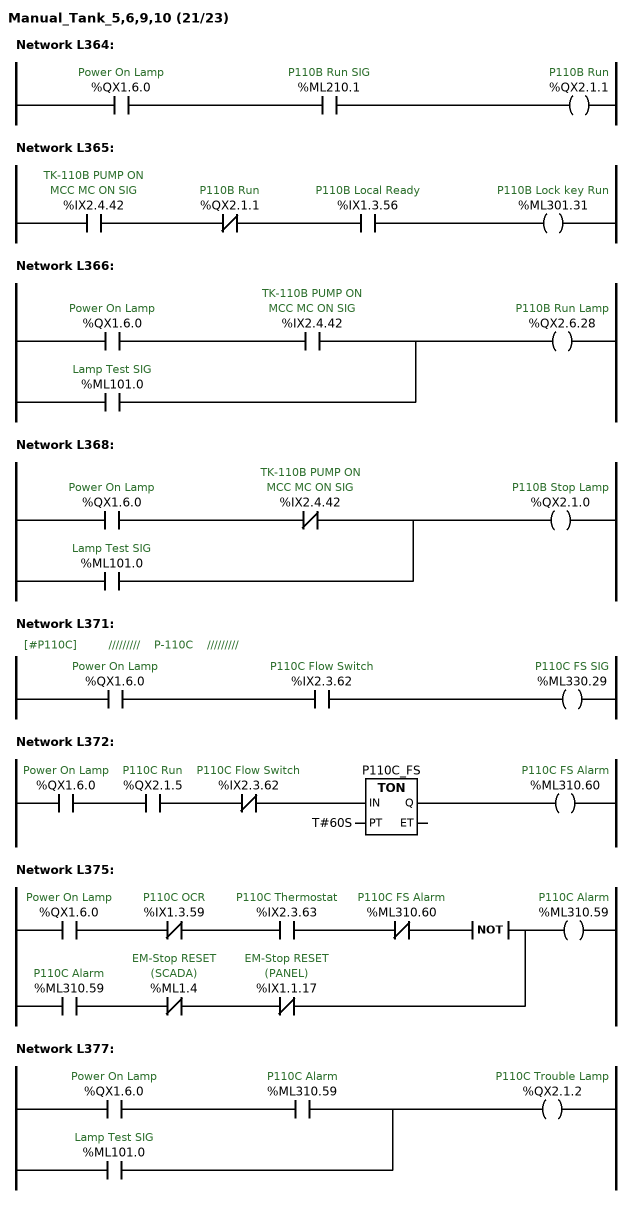
(* [picture p72: Manual_Tank_5,6,9,10 rungs L364-L377] *)
(* Rung L364 *)
%QX2.1.1 := %QX1.6.0 AND %ML210.1;
(* Rung L365 *)
%ML301.31 := %IX2.4.42 AND NOT %QX2.1.1 AND %IX1.3.56;
(* Rung L366 *)
%QX2.6.28 := (%QX1.6.0 AND %IX2.4.42) OR %ML101.0;
(* Rung L368 *)
%QX2.1.0 := (%QX1.6.0 AND NOT %IX2.4.42) OR %ML101.0;
(* [#P110C]         /////////    P-110C    ///////// *)
(* Rung L371 *)
%ML330.29 := %QX1.6.0 AND %IX2.3.62;
(* Rung L372 *)
P110C_FS(IN := %QX1.6.0 AND %QX2.1.5 AND NOT %IX2.3.62, PT := T#60S);
%ML310.60 := P110C_FS.Q;
(* Rung L375 *)
%ML310.59 := NOT (%QX1.6.0 AND NOT %IX1.3.59 AND %IX2.3.63 AND NOT %ML310.60) OR (%ML310.59 AND NOT %ML1.4 AND NOT %IX1.1.17);
(* Rung L377 *)
%QX2.1.2 := (%QX1.6.0 AND %ML310.59) OR %ML101.0;

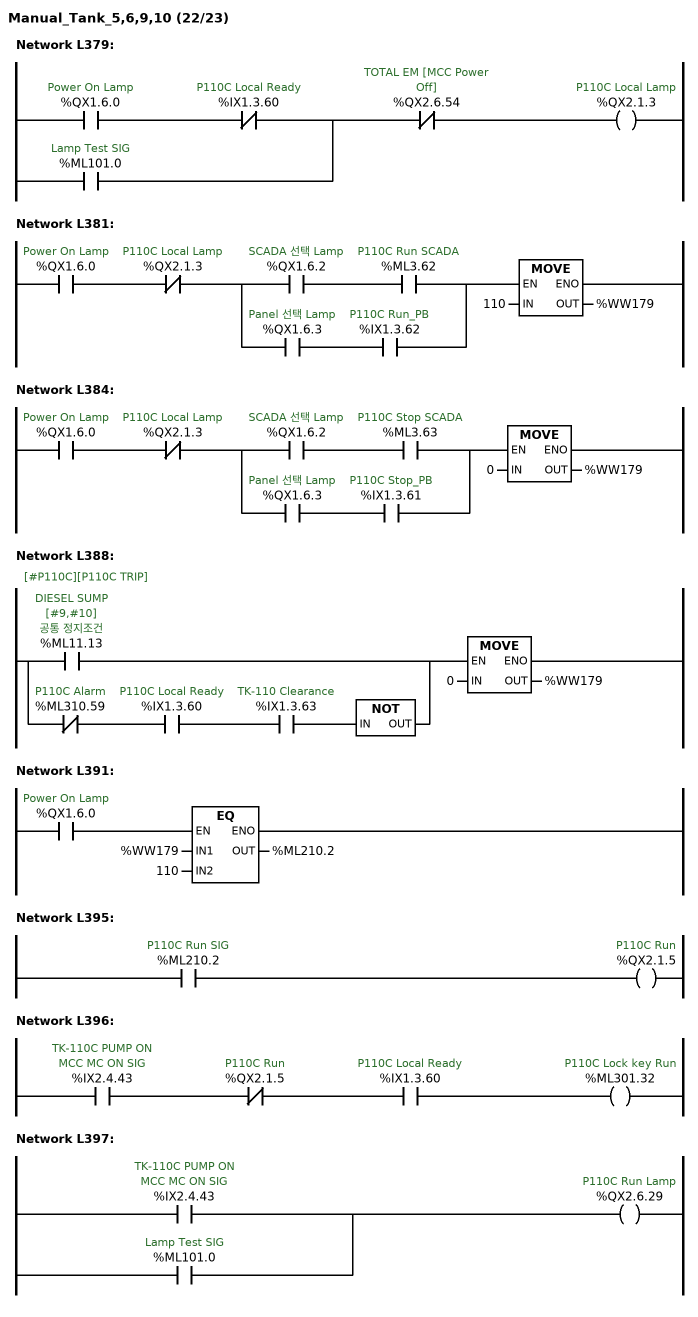
(* Rung L379 *)
%QX2.1.3 := ((%QX1.6.0 AND NOT %IX1.3.60) OR %ML101.0) AND NOT %QX2.6.54;
(* Rung L381 *)
IF %QX1.6.0 AND NOT %QX2.1.3 AND ((%QX1.6.2 AND %ML3.62) OR (%QX1.6.3 AND %IX1.3.62)) THEN
    %WW179 := 110;
END_IF;
(* Rung L384 *)
IF %QX1.6.0 AND NOT %QX2.1.3 AND ((%QX1.6.2 AND %ML3.63) OR (%QX1.6.3 AND %IX1.3.61)) THEN
    %WW179 := 0;
END_IF;
(* [#P110C][P110C TRIP] *)
(* Rung L388 *)
IF %ML11.13 OR (NOT (NOT %ML310.59 AND %IX1.3.60 AND %IX1.3.63)) THEN %WW179 := 0; END_IF;
(* Rung L391 *)
IF %QX1.6.0 THEN %ML210.2 := %WW179 = 110; END_IF;
(* Rung L395 *)
%QX2.1.5 := %ML210.2;
(* Rung L396 *)
%ML301.32 := %IX2.4.43 AND NOT %QX2.1.5 AND %IX1.3.60;
(* Rung L397 *)
%QX2.6.29 := %IX2.4.43 OR %ML101.0;

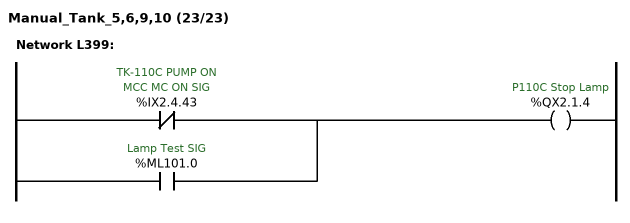
(* Rung L399 *)
%QX2.1.4 := NOT %IX2.4.43 OR %ML101.0;
END_PROGRAM

PROGRAM Manual_Drain_Tank (* task: 스캔 프로그램 *)
VAR
    TK_111_FS : TON;
    TK_112_FS : TON;
    TK_113_FS : TON;
END_VAR

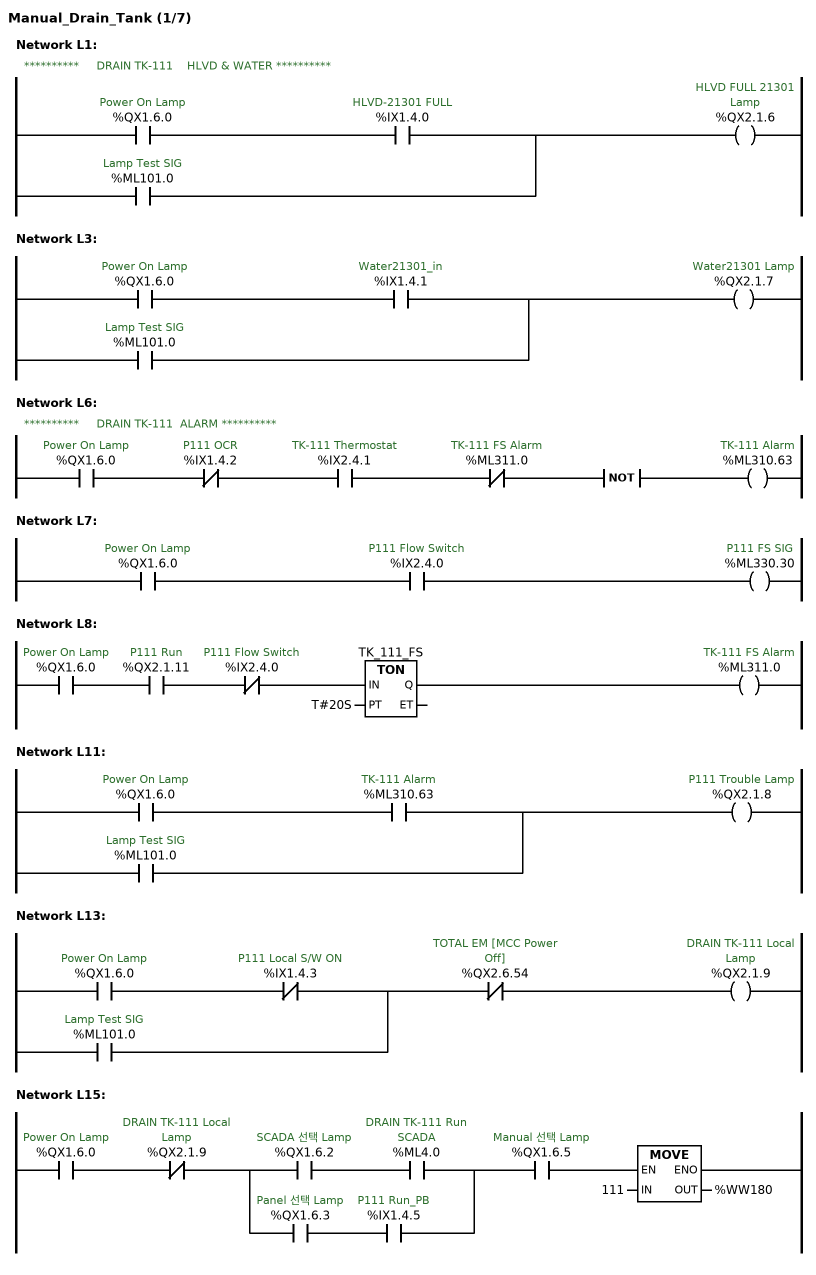
(* **********     DRAIN TK-111    HLVD & WATER ********** *)
(* Rung L1 *)
%QX2.1.6 := (%QX1.6.0 AND %IX1.4.0) OR %ML101.0;
(* Rung L3 *)
%QX2.1.7 := (%QX1.6.0 AND %IX1.4.1) OR %ML101.0;
(* **********     DRAIN TK-111  ALARM ********** *)
(* Rung L6 *)
%ML310.63 := NOT (%QX1.6.0 AND NOT %IX1.4.2 AND %IX2.4.1 AND NOT %ML311.0);
(* Rung L7 *)
%ML330.30 := %QX1.6.0 AND %IX2.4.0;
(* Rung L8 *)
TK_111_FS(IN := %QX1.6.0 AND %QX2.1.11 AND NOT %IX2.4.0, PT := T#20S);
%ML311.0 := TK_111_FS.Q;
(* Rung L11 *)
%QX2.1.8 := (%QX1.6.0 AND %ML310.63) OR %ML101.0;
(* Rung L13 *)
%QX2.1.9 := ((%QX1.6.0 AND NOT %IX1.4.3) OR %ML101.0) AND NOT %QX2.6.54;
(* Rung L15 *)
IF %QX1.6.0 AND NOT %QX2.1.9 AND ((%QX1.6.2 AND %ML4.0) OR (%QX1.6.3 AND %IX1.4.5)) AND %QX1.6.5 THEN
    %WW180 := 111;
END_IF;

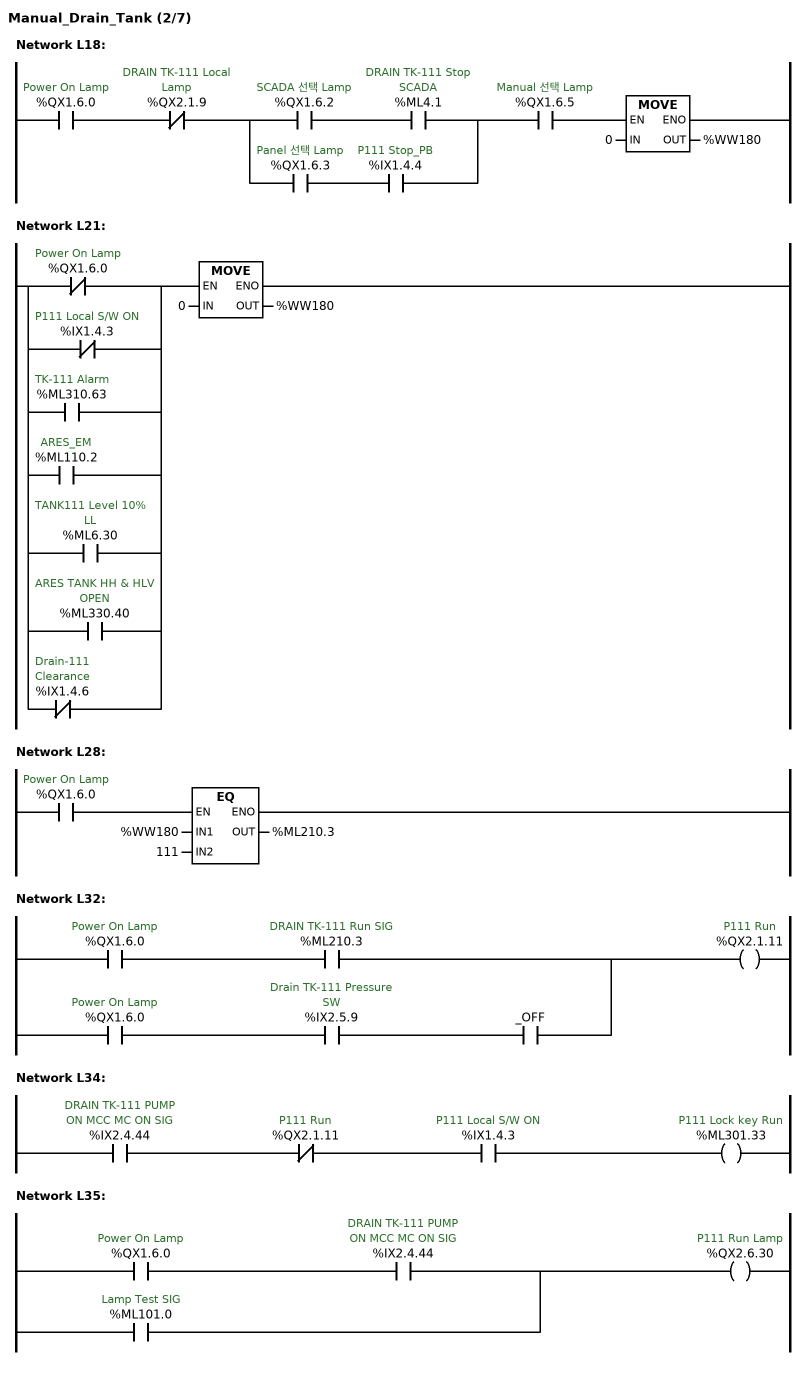
(* Rung L18 *)
IF %QX1.6.0 AND NOT %QX2.1.9 AND ((%QX1.6.2 AND %ML4.1) OR (%QX1.6.3 AND %IX1.4.4)) AND %QX1.6.5 THEN
    %WW180 := 0;
END_IF;
(* Rung L21 *)
IF NOT %QX1.6.0 OR NOT %IX1.4.3 OR %ML310.63 OR %ML110.2 OR %ML6.30 OR %ML330.40 OR NOT %IX1.4.6 THEN
    %WW180 := 0;
END_IF;
(* Rung L28 *)
IF %QX1.6.0 THEN %ML210.3 := %WW180 = 111; END_IF;
(* Rung L32 *)
%QX2.1.11 := (%QX1.6.0 AND %ML210.3) OR (%QX1.6.0 AND %IX2.5.9 AND _OFF);
(* Rung L34 *)
%ML301.33 := %IX2.4.44 AND NOT %QX2.1.11 AND %IX1.4.3;
(* Rung L35 *)
%QX2.6.30 := (%QX1.6.0 AND %IX2.4.44) OR %ML101.0;

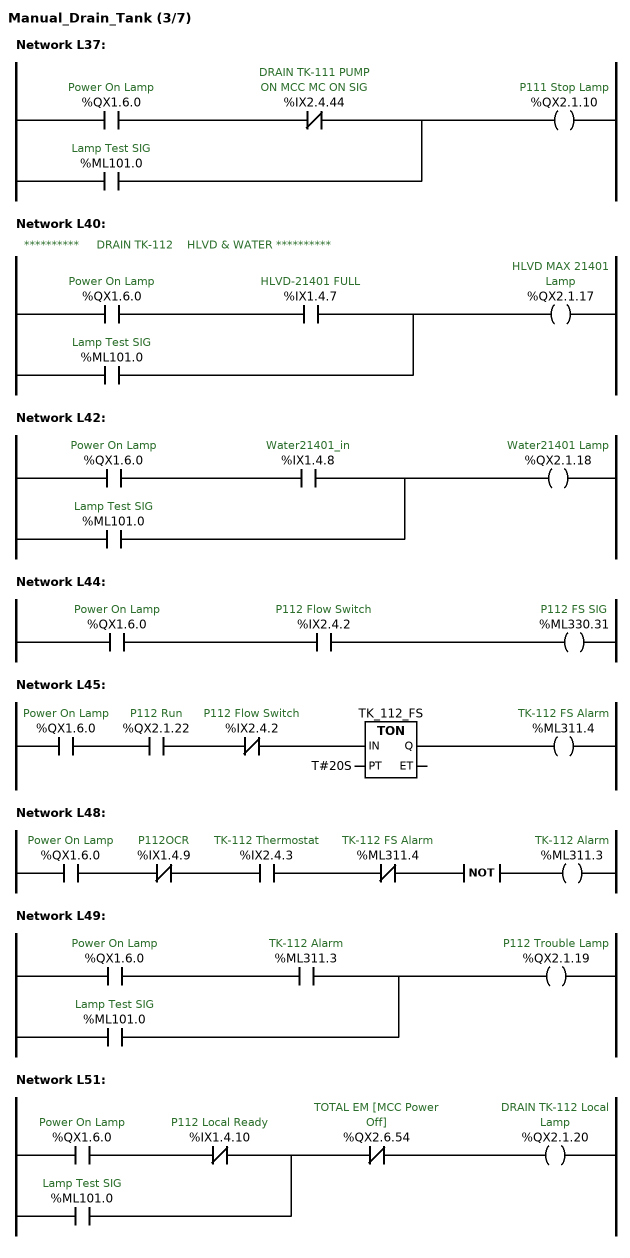
(* Rung L37 *)
%QX2.1.10 := (%QX1.6.0 AND NOT %IX2.4.44) OR %ML101.0;
(* **********     DRAIN TK-112    HLVD & WATER ********** *)
(* Rung L40 *)
%QX2.1.17 := (%QX1.6.0 AND %IX1.4.7) OR %ML101.0;
(* Rung L42 *)
%QX2.1.18 := (%QX1.6.0 AND %IX1.4.8) OR %ML101.0;
(* Rung L44 *)
%ML330.31 := %QX1.6.0 AND %IX2.4.2;
(* Rung L45 *)
TK_112_FS(IN := %QX1.6.0 AND %QX2.1.22 AND NOT %IX2.4.2, PT := T#20S);
%ML311.4 := TK_112_FS.Q;
(* Rung L48 *)
%ML311.3 := NOT (%QX1.6.0 AND NOT %IX1.4.9 AND %IX2.4.3 AND NOT %ML311.4);
(* Rung L49 *)
%QX2.1.19 := (%QX1.6.0 AND %ML311.3) OR %ML101.0;
(* Rung L51 *)
%QX2.1.20 := ((%QX1.6.0 AND NOT %IX1.4.10) OR %ML101.0) AND NOT %QX2.6.54;

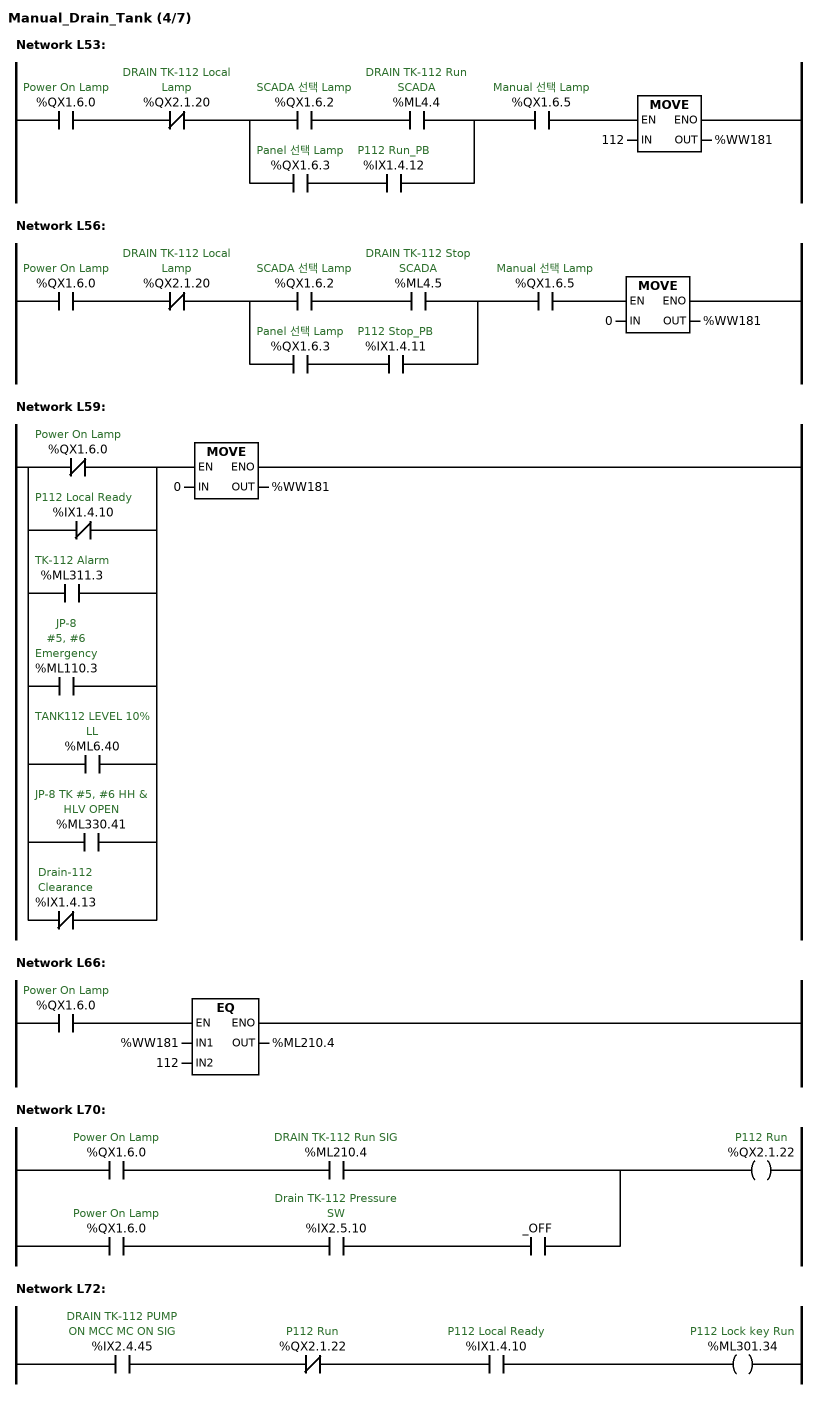
(* Rung L53 *)
IF %QX1.6.0 AND NOT %QX2.1.20 AND ((%QX1.6.2 AND %ML4.4) OR (%QX1.6.3 AND %IX1.4.12)) AND %QX1.6.5 THEN
    %WW181 := 112;
END_IF;
(* Rung L56 *)
IF %QX1.6.0 AND NOT %QX2.1.20 AND ((%QX1.6.2 AND %ML4.5) OR (%QX1.6.3 AND %IX1.4.11)) AND %QX1.6.5 THEN
    %WW181 := 0;
END_IF;
(* Rung L59 *)
IF NOT %QX1.6.0 OR NOT %IX1.4.10 OR %ML311.3 OR %ML110.3 OR %ML6.40 OR %ML330.41 OR NOT %IX1.4.13 THEN
    %WW181 := 0;
END_IF;
(* Rung L66 *)
IF %QX1.6.0 THEN %ML210.4 := %WW181 = 112; END_IF;
(* Rung L70 *)
%QX2.1.22 := (%QX1.6.0 AND %ML210.4) OR (%QX1.6.0 AND %IX2.5.10 AND _OFF);
(* Rung L72 *)
%ML301.34 := %IX2.4.45 AND NOT %QX2.1.22 AND %IX1.4.10;

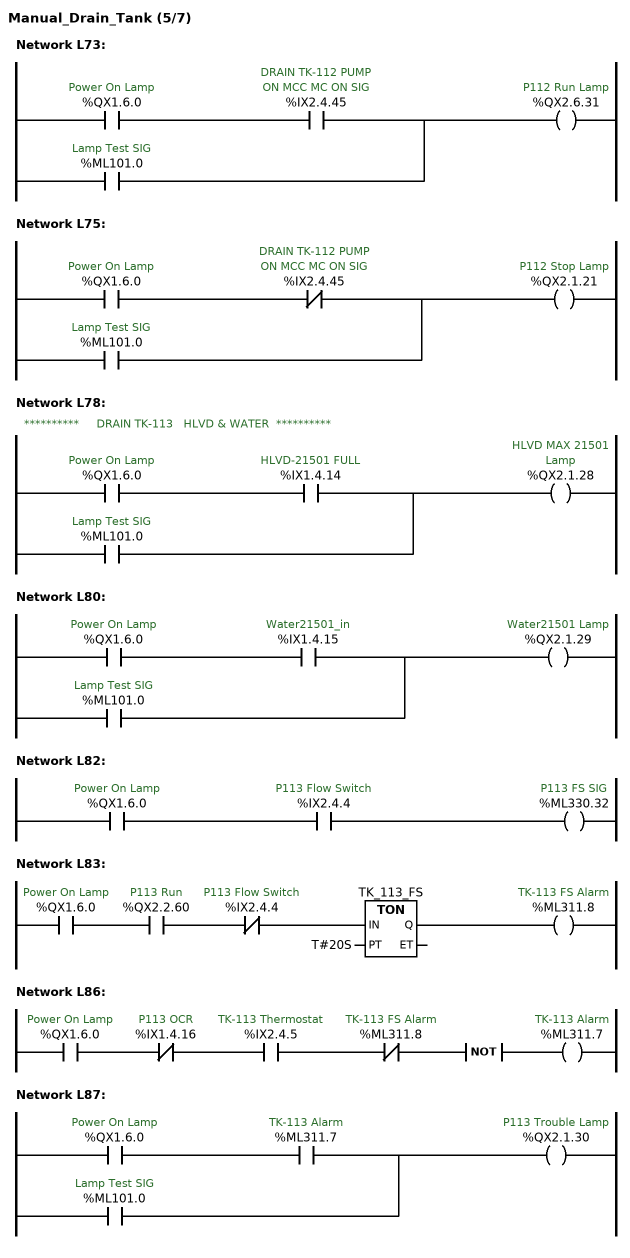
(* Rung L73 *)
%QX2.6.31 := (%QX1.6.0 AND %IX2.4.45) OR %ML101.0;
(* Rung L75 *)
%QX2.1.21 := (%QX1.6.0 AND NOT %IX2.4.45) OR %ML101.0;
(* **********     DRAIN TK-113   HLVD & WATER  ********** *)
(* Rung L78 *)
%QX2.1.28 := (%QX1.6.0 AND %IX1.4.14) OR %ML101.0;
(* Rung L80 *)
%QX2.1.29 := (%QX1.6.0 AND %IX1.4.15) OR %ML101.0;
(* Rung L82 *)
%ML330.32 := %QX1.6.0 AND %IX2.4.4;
(* Rung L83 *)
TK_113_FS(IN := %QX1.6.0 AND %QX2.2.60 AND NOT %IX2.4.4, PT := T#20S);
%ML311.8 := TK_113_FS.Q;
(* Rung L86 *)
%ML311.7 := NOT (%QX1.6.0 AND NOT %IX1.4.16 AND %IX2.4.5 AND NOT %ML311.8);
(* Rung L87 *)
%QX2.1.30 := (%QX1.6.0 AND %ML311.7) OR %ML101.0;

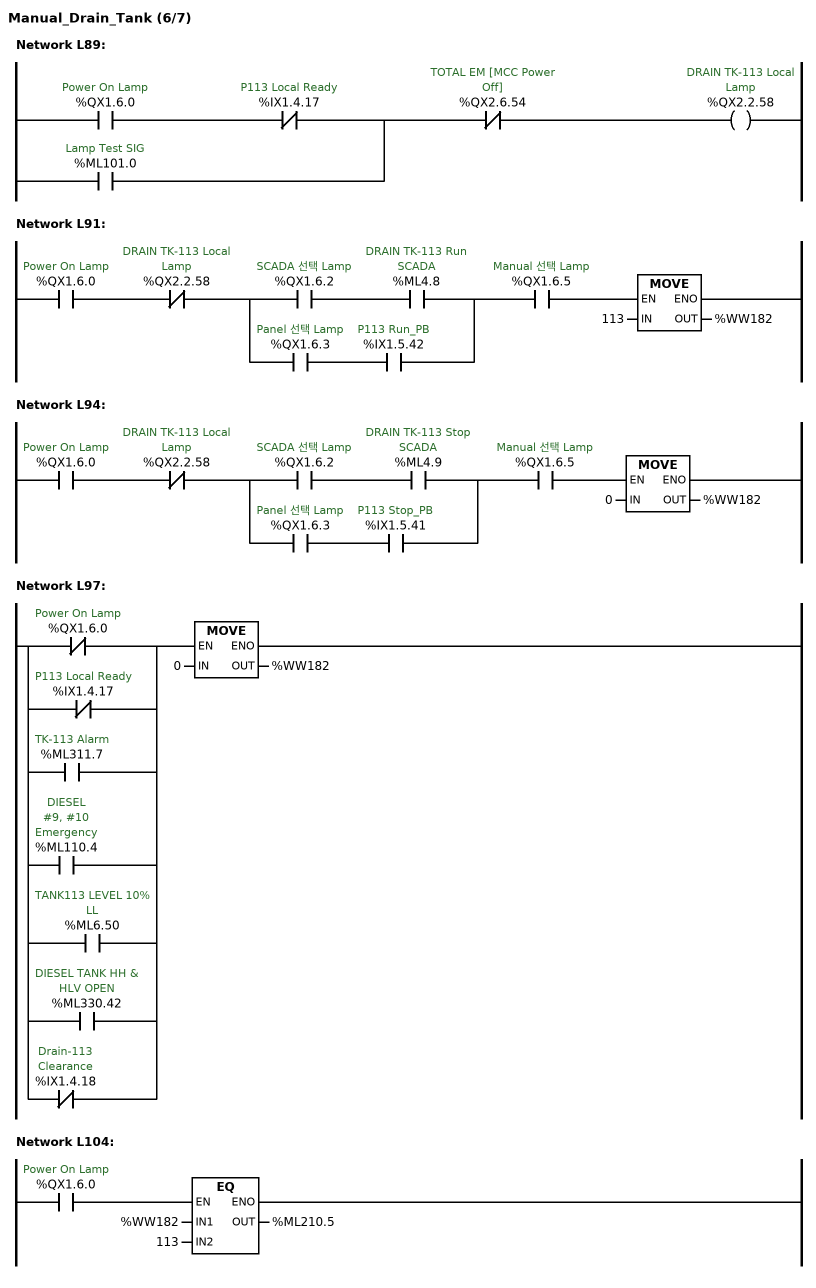
(* Rung L89 *)
%QX2.2.58 := ((%QX1.6.0 AND NOT %IX1.4.17) OR %ML101.0) AND NOT %QX2.6.54;
(* Rung L91 *)
IF %QX1.6.0 AND NOT %QX2.2.58 AND ((%QX1.6.2 AND %ML4.8) OR (%QX1.6.3 AND %IX1.5.42)) AND %QX1.6.5 THEN
    %WW182 := 113;
END_IF;
(* Rung L94 *)
IF %QX1.6.0 AND NOT %QX2.2.58 AND ((%QX1.6.2 AND %ML4.9) OR (%QX1.6.3 AND %IX1.5.41)) AND %QX1.6.5 THEN
    %WW182 := 0;
END_IF;
(* Rung L97 *)
IF NOT %QX1.6.0 OR NOT %IX1.4.17 OR %ML311.7 OR %ML110.4 OR %ML6.50 OR %ML330.42 OR NOT %IX1.4.18 THEN
    %WW182 := 0;
END_IF;
(* Rung L104 *)
IF %QX1.6.0 THEN %ML210.5 := %WW182 = 113; END_IF;

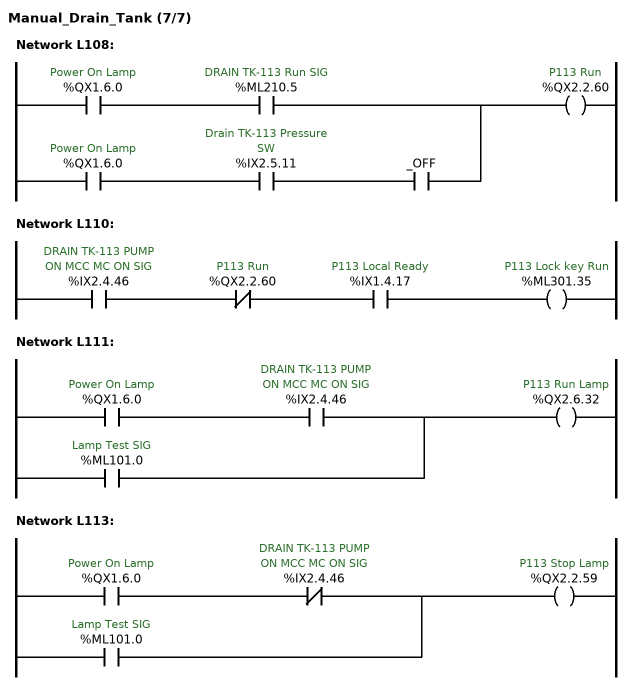
(* Rung L108 *)
%QX2.2.60 := (%QX1.6.0 AND %ML210.5) OR (%QX1.6.0 AND %IX2.5.11 AND _OFF);
(* Rung L110 *)
%ML301.35 := %IX2.4.46 AND NOT %QX2.2.60 AND %IX1.4.17;
(* Rung L111 *)
%QX2.6.32 := (%QX1.6.0 AND %IX2.4.46) OR %ML101.0;
(* Rung L113 *)
%QX2.2.59 := (%QX1.6.0 AND NOT %IX2.4.46) OR %ML101.0;
END_PROGRAM

PROGRAM Manual_Mov (* task: 스캔 프로그램 *)
VAR
    _p1 : BOOL;
    _p2 : BOOL;
    _p3 : BOOL;
END_VAR

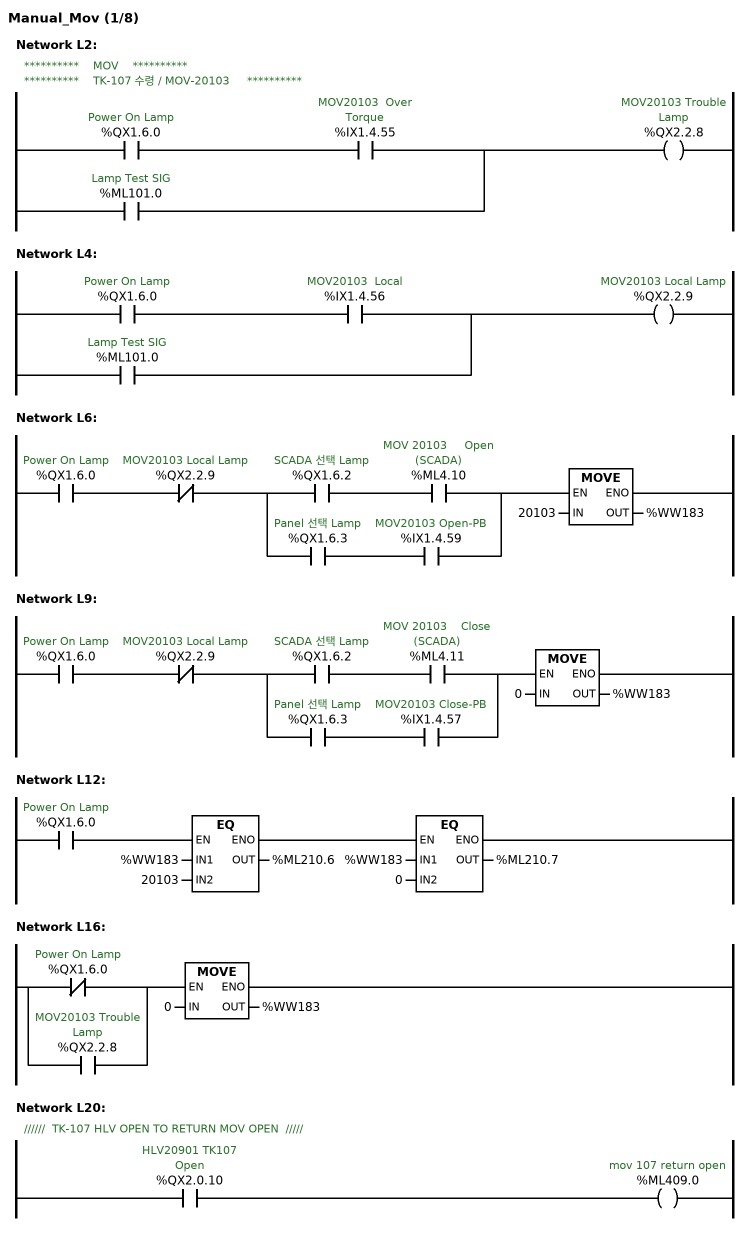
(* **********    MOV    ********** *)
(* **********    TK-107 수령 / MOV-20103     ********** *)
(* Rung L2 *)
%QX2.2.8 := (%QX1.6.0 AND %IX1.4.55) OR %ML101.0;
(* Rung L4 *)
%QX2.2.9 := (%QX1.6.0 AND %IX1.4.56) OR %ML101.0;
(* Rung L6 *)
IF %QX1.6.0 AND NOT %QX2.2.9 AND ((%QX1.6.2 AND %ML4.10) OR (%QX1.6.3 AND %IX1.4.59)) THEN
    %WW183 := 20103;
END_IF;
(* Rung L9 *)
IF %QX1.6.0 AND NOT %QX2.2.9 AND ((%QX1.6.2 AND %ML4.11) OR (%QX1.6.3 AND %IX1.4.57)) THEN
    %WW183 := 0;
END_IF;
(* Rung L12 *)
IF %QX1.6.0 THEN
    %ML210.6 := %WW183 = 20103;
    %ML210.7 := %WW183 = 0;
END_IF;
(* Rung L16 *)
IF NOT %QX1.6.0 OR %QX2.2.8 THEN %WW183 := 0; END_IF;
(* //////  TK-107 HLV OPEN TO RETURN MOV OPEN  ///// *)
(* Rung L20 *)
%ML409.0 := %QX2.0.10;

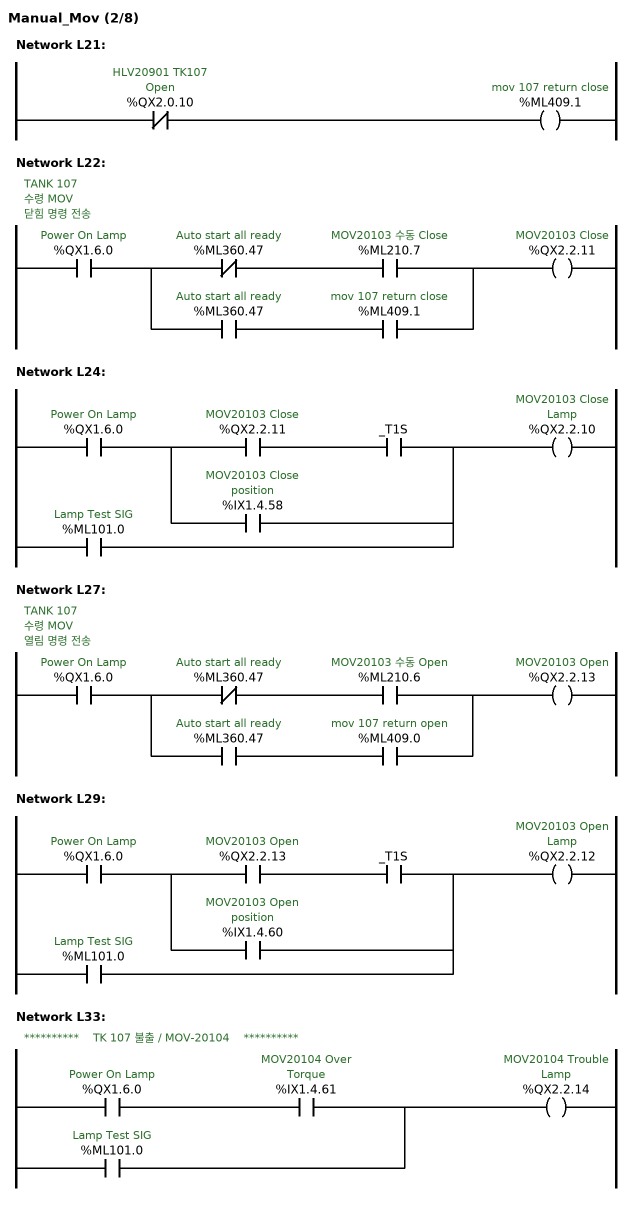
(* Rung L21 *)
%ML409.1 := NOT %QX2.0.10;
(* Rung L22 *)
%QX2.2.11 := %QX1.6.0 AND ((NOT %ML360.47 AND %ML210.7) OR (%ML360.47 AND %ML409.1));
(* TANK 107 / 수령 MOV / 닫힘 명령 전송 *)
(* Rung L24 *)
%QX2.2.10 := (%QX1.6.0 AND ((%QX2.2.11 AND _T1S) OR %IX1.4.58)) OR %ML101.0;
(* Rung L27 *)
%QX2.2.13 := %QX1.6.0 AND ((NOT %ML360.47 AND %ML210.6) OR (%ML360.47 AND %ML409.0));
(* TANK 107 / 수령 MOV / 열림 명령 전송 *)
(* Rung L29 *)
%QX2.2.12 := (%QX1.6.0 AND ((%QX2.2.13 AND _T1S) OR %IX1.4.60)) OR %ML101.0;
(* **********    TK 107 불출 / MOV-20104    ********** *)
(* Rung L33 *)
%QX2.2.14 := (%QX1.6.0 AND %IX1.4.61) OR %ML101.0;

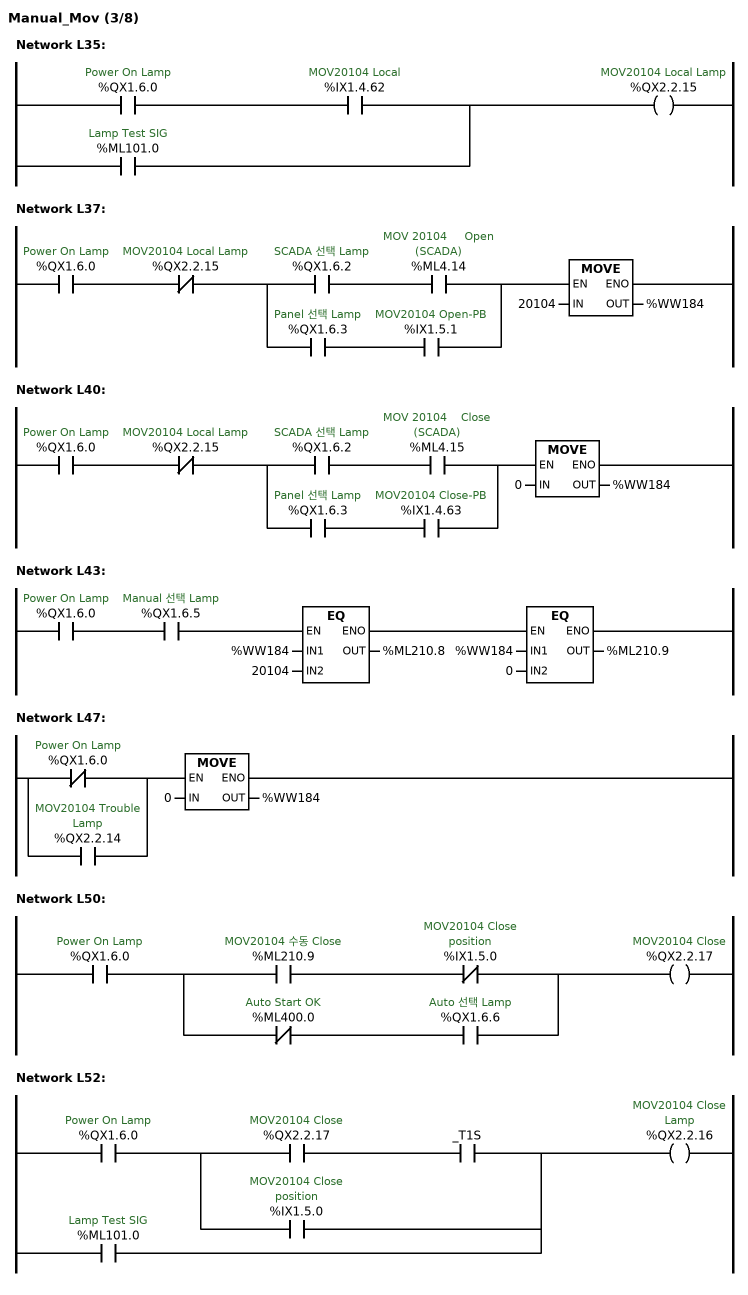
(* Rung L35 *)
%QX2.2.15 := (%QX1.6.0 AND %IX1.4.62) OR %ML101.0;
(* Rung L37 *)
IF %QX1.6.0 AND NOT %QX2.2.15 AND ((%QX1.6.2 AND %ML4.14) OR (%QX1.6.3 AND %IX1.5.1)) THEN
    %WW184 := 20104;
END_IF;
(* Rung L40 *)
IF %QX1.6.0 AND NOT %QX2.2.15 AND ((%QX1.6.2 AND %ML4.15) OR (%QX1.6.3 AND %IX1.4.63)) THEN
    %WW184 := 0;
END_IF;
(* Rung L43 *)
IF %QX1.6.0 AND %QX1.6.5 THEN
    %ML210.8 := %WW184 = 20104;
    %ML210.9 := %WW184 = 0;
END_IF;
(* Rung L47 *)
IF NOT %QX1.6.0 OR %QX2.2.14 THEN %WW184 := 0; END_IF;
(* Rung L50 *)
%QX2.2.17 := %QX1.6.0 AND ((%ML210.9 AND NOT %IX1.5.0) OR (NOT %ML400.0 AND %QX1.6.6));
(* Rung L52 *)
%QX2.2.16 := (%QX1.6.0 AND ((%QX2.2.17 AND _T1S) OR %IX1.5.0)) OR %ML101.0;

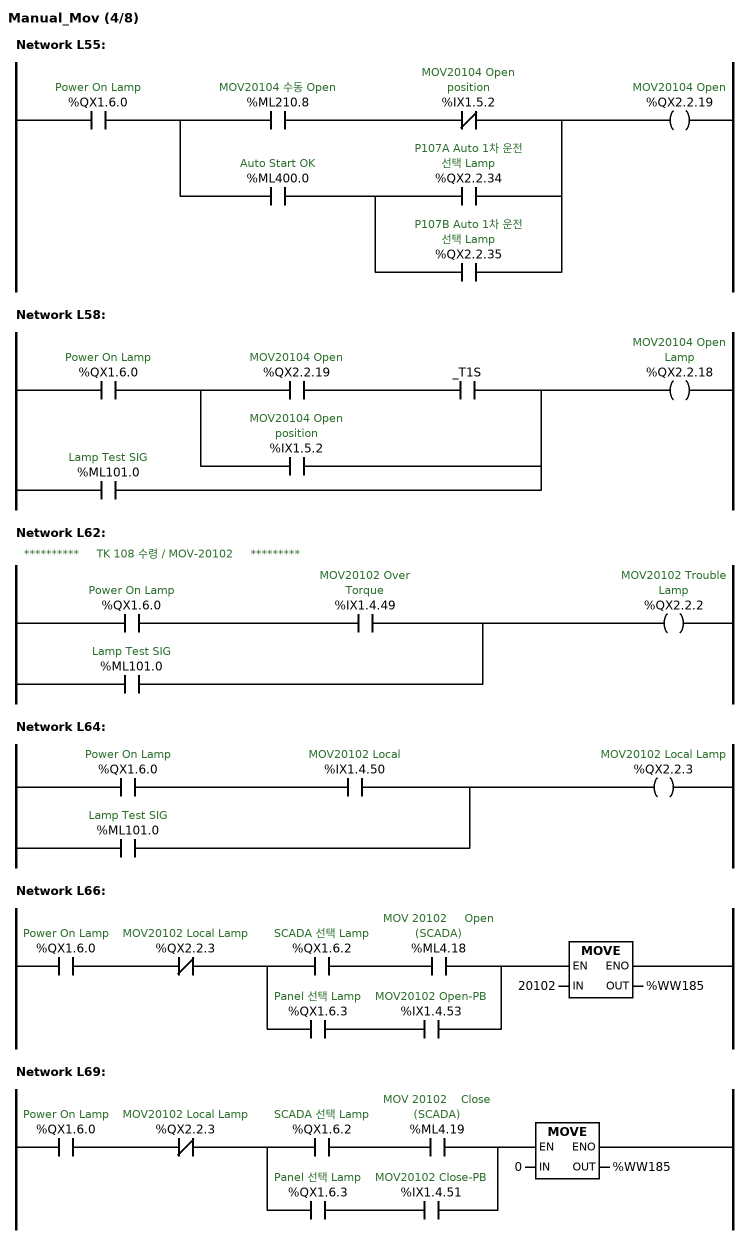
(* Rung L55 *)
%QX2.2.19 := %QX1.6.0 AND ((%ML210.8 AND NOT %IX1.5.2) OR (%ML400.0 AND (%QX2.2.34 OR %QX2.2.35)));
(* Rung L58 *)
%QX2.2.18 := (%QX1.6.0 AND ((%QX2.2.19 AND _T1S) OR %IX1.5.2)) OR %ML101.0;
(* **********     TK 108 수령 / MOV-20102     ********* *)
(* Rung L62 *)
%QX2.2.2 := (%QX1.6.0 AND %IX1.4.49) OR %ML101.0;
(* Rung L64 *)
%QX2.2.3 := (%QX1.6.0 AND %IX1.4.50) OR %ML101.0;
(* Rung L66 *)
IF %QX1.6.0 AND NOT %QX2.2.3 AND ((%QX1.6.2 AND %ML4.18) OR (%QX1.6.3 AND %IX1.4.53)) THEN
    %WW185 := 20102;
END_IF;
(* Rung L69 *)
IF %QX1.6.0 AND NOT %QX2.2.3 AND ((%QX1.6.2 AND %ML4.19) OR (%QX1.6.3 AND %IX1.4.51)) THEN
    %WW185 := 0;
END_IF;

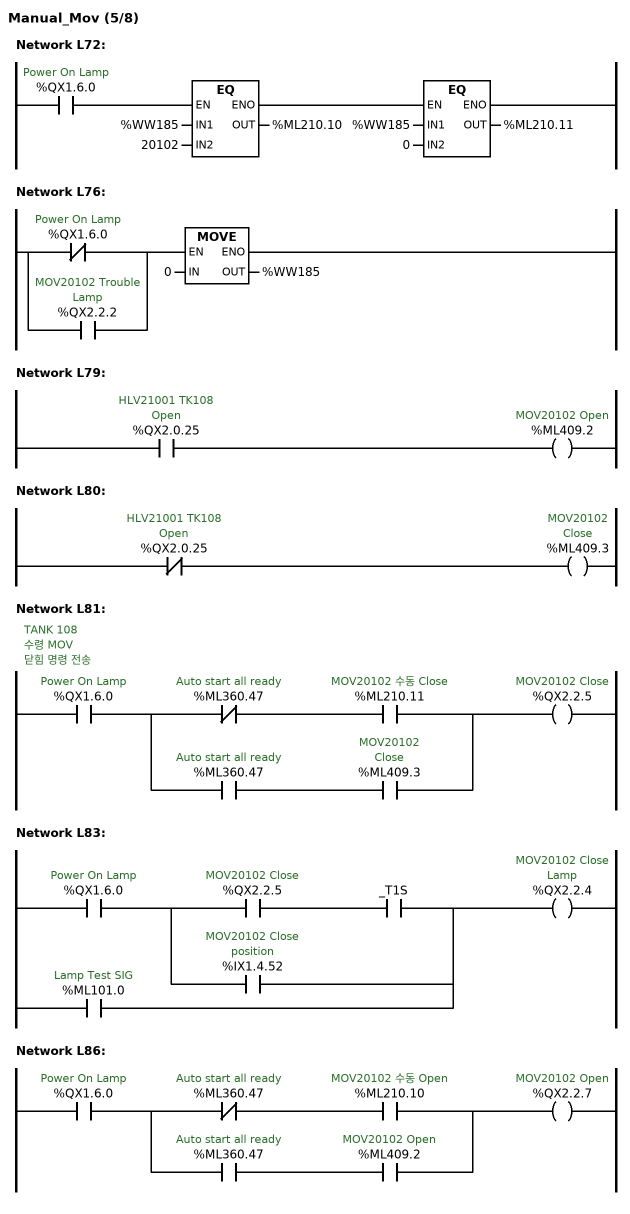
(* Rung L72 *)
IF %QX1.6.0 THEN
    %ML210.10 := %WW185 = 20102;
    %ML210.11 := %WW185 = 0;
END_IF;
(* Rung L76 *)
IF NOT %QX1.6.0 OR %QX2.2.2 THEN %WW185 := 0; END_IF;
(* Rung L79 *)
%ML409.2 := %QX2.0.25;
(* Rung L80 *)
%ML409.3 := NOT %QX2.0.25;
(* Rung L81 *)
%QX2.2.5 := %QX1.6.0 AND ((NOT %ML360.47 AND %ML210.11) OR (%ML360.47 AND %ML409.3));
(* TANK 108 / 수령 MOV / 닫힘 명령 전송 *)
(* Rung L83 *)
%QX2.2.4 := (%QX1.6.0 AND ((%QX2.2.5 AND _T1S) OR %IX1.4.52)) OR %ML101.0;
(* Rung L86 *)
%QX2.2.7 := %QX1.6.0 AND ((NOT %ML360.47 AND %ML210.10) OR (%ML360.47 AND %ML409.2));

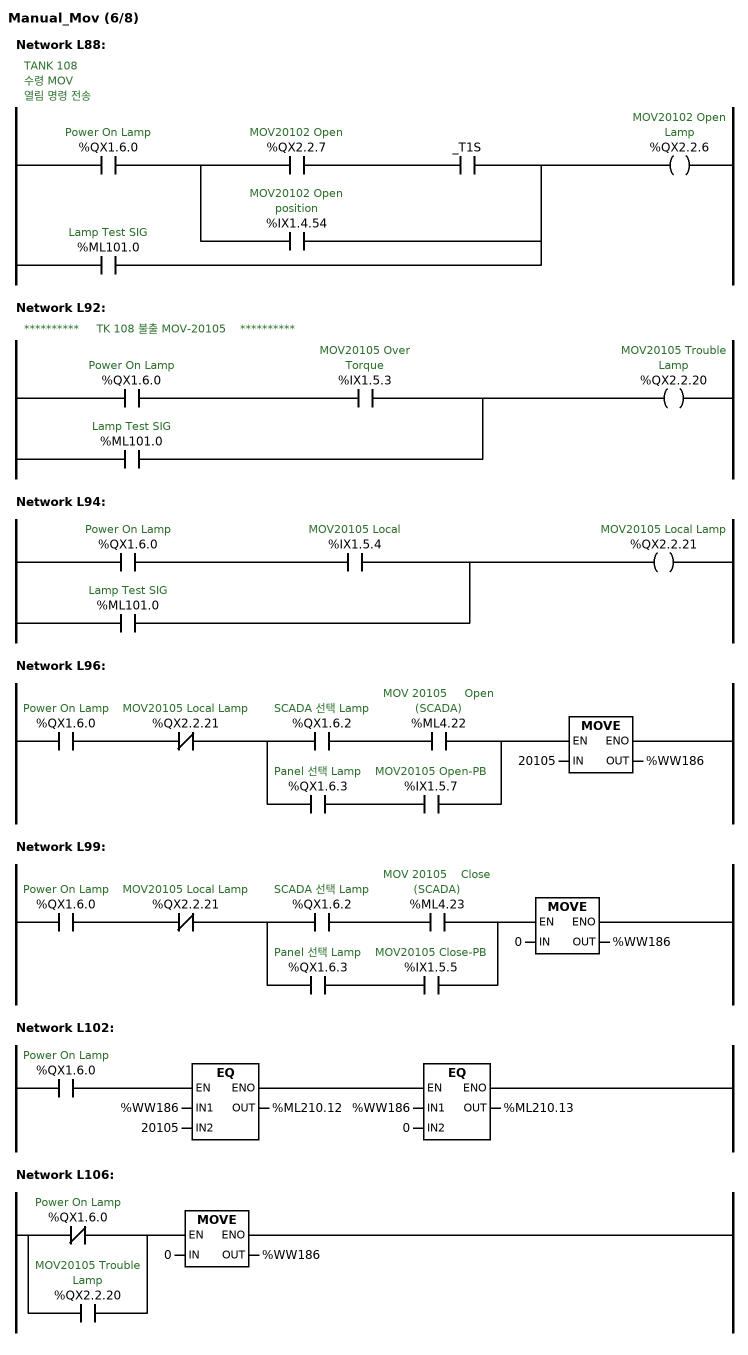
(* Rung L88 *)
%QX2.2.6 := (%QX1.6.0 AND ((%QX2.2.7 AND _T1S) OR %IX1.4.54)) OR %ML101.0;
(* TANK 108 / 수령 MOV / 열림 명령 전송 *)
(* **********     TK 108 불출 MOV-20105    ********** *)
(* Rung L92 *)
%QX2.2.20 := (%QX1.6.0 AND %IX1.5.3) OR %ML101.0;
(* Rung L94 *)
%QX2.2.21 := (%QX1.6.0 AND %IX1.5.4) OR %ML101.0;
(* Rung L96 *)
IF %QX1.6.0 AND NOT %QX2.2.21 AND ((%QX1.6.2 AND %ML4.22) OR (%QX1.6.3 AND %IX1.5.7)) THEN
    %WW186 := 20105;
END_IF;
(* Rung L99 *)
IF %QX1.6.0 AND NOT %QX2.2.21 AND ((%QX1.6.2 AND %ML4.23) OR (%QX1.6.3 AND %IX1.5.5)) THEN
    %WW186 := 0;
END_IF;
(* Rung L102 *)
IF %QX1.6.0 THEN
    %ML210.12 := %WW186 = 20105;
    %ML210.13 := %WW186 = 0;
END_IF;
(* Rung L106 *)
IF NOT %QX1.6.0 OR %QX2.2.20 THEN %WW186 := 0; END_IF;

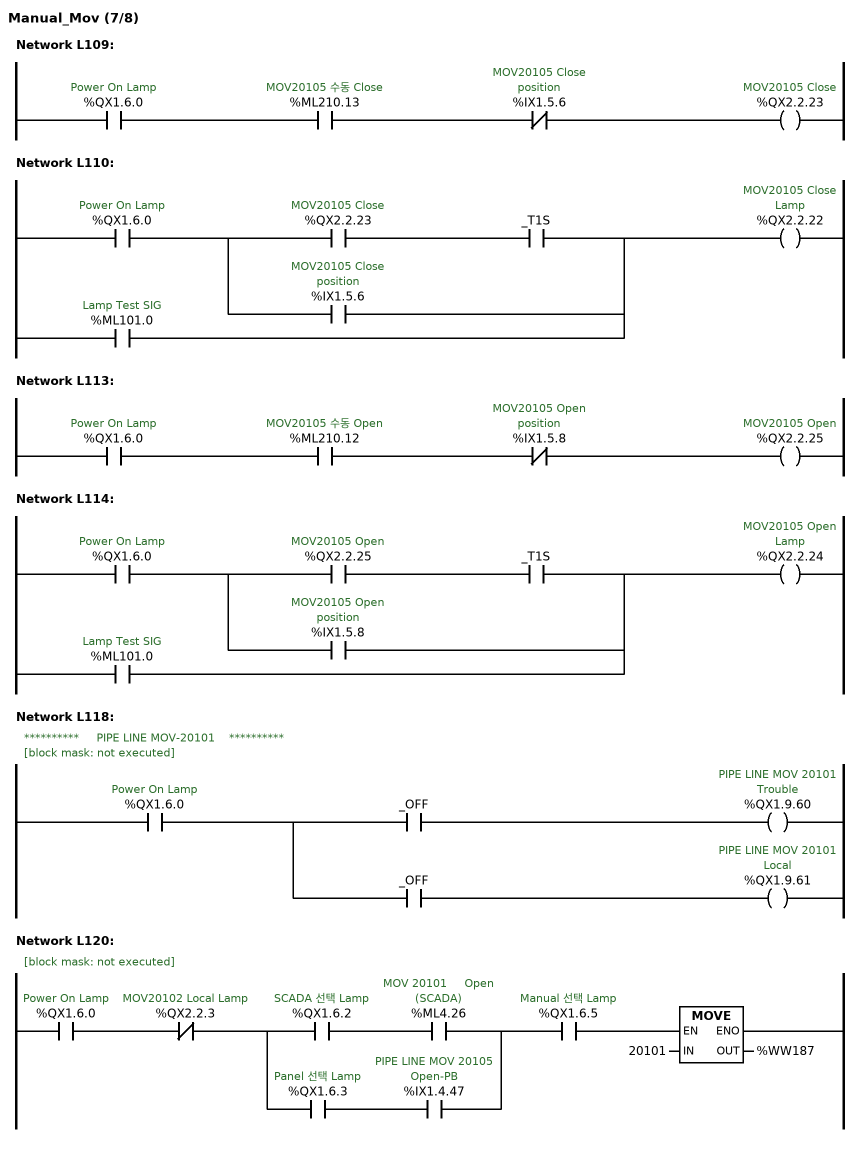
(* Rung L109 *)
%QX2.2.23 := %QX1.6.0 AND %ML210.13 AND NOT %IX1.5.6;
(* Rung L110 *)
%QX2.2.22 := (%QX1.6.0 AND ((%QX2.2.23 AND _T1S) OR %IX1.5.6)) OR %ML101.0;
(* Rung L113 *)
%QX2.2.25 := %QX1.6.0 AND %ML210.12 AND NOT %IX1.5.8;
(* Rung L114 *)
%QX2.2.24 := (%QX1.6.0 AND ((%QX2.2.25 AND _T1S) OR %IX1.5.8)) OR %ML101.0;
(* **********     PIPE LINE MOV-20101    ********** *)
(* Rung L118 is block-masked: not executed *)
// _p1 := %QX1.6.0;
// %QX1.9.60 := %QX1.6.0 AND _OFF;
// %QX1.9.61 := _p1 AND _OFF;
(* Rung L120 is block-masked: not executed *)
// IF %QX1.6.0 AND NOT %QX2.2.3 AND ((%QX1.6.2 AND %ML4.26) OR (%QX1.6.3 AND %IX1.4.47)) AND %QX1.6.5 THEN
//     %WW187 := 20101;
// END_IF;

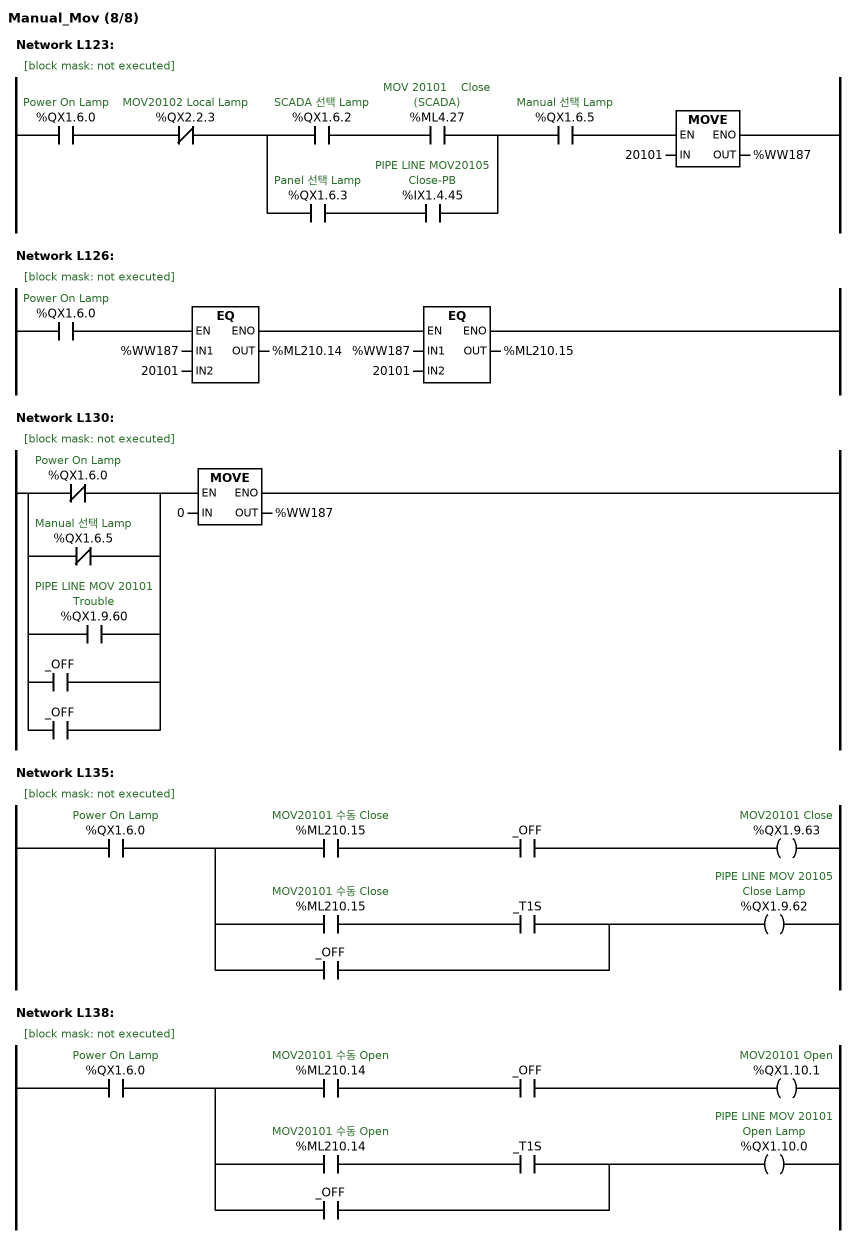
(* Rung L123 is block-masked: not executed *)
// IF %QX1.6.0 AND NOT %QX2.2.3 AND ((%QX1.6.2 AND %ML4.27) OR (%QX1.6.3 AND %IX1.4.45)) AND %QX1.6.5 THEN
//     %WW187 := 20101;
// END_IF;
(* Rung L126 is block-masked: not executed *)
// IF %QX1.6.0 THEN
//     %ML210.14 := %WW187 = 20101;
//     %ML210.15 := %WW187 = 20101;
// END_IF;
(* Rung L130 is block-masked: not executed *)
// IF NOT %QX1.6.0 OR NOT %QX1.6.5 OR %QX1.9.60 OR _OFF OR _OFF THEN %WW187 := 0; END_IF;
(* Rung L135 is block-masked: not executed *)
// _p2 := %QX1.6.0;
// %QX1.9.63 := %QX1.6.0 AND %ML210.15 AND _OFF;
// %QX1.9.62 := _p2 AND ((%ML210.15 AND _T1S) OR _OFF);
(* Rung L138 is block-masked: not executed *)
// _p3 := %QX1.6.0;
// %QX1.10.1 := %QX1.6.0 AND %ML210.14 AND _OFF;
// %QX1.10.0 := _p3 AND ((%ML210.14 AND _T1S) OR _OFF);
END_PROGRAM

PROGRAM Manual_Unlodang_Pump (* task: 스캔 프로그램 *)
VAR
    TK_111_FS : TON;
    UP201A_FS : TON; (* UP102A_FS ALARM DELAY TIME *)
    UP201B_FS : TON;
    UP202A_FS : TON; (* UP102A_FS ALARM DELAY TIME *)
    UP202B_FS : TON;
    UP203A_FS : TON;
    UP203A_FS_TON : TON; (* P203A FLOW SWITCH ALARM DELAY TIMER *)
    UP203B_FS : TON;
    UP204A_FS : TON;
    UP204B_FS : TON;
    UP205B_FS : TON;
END_VAR

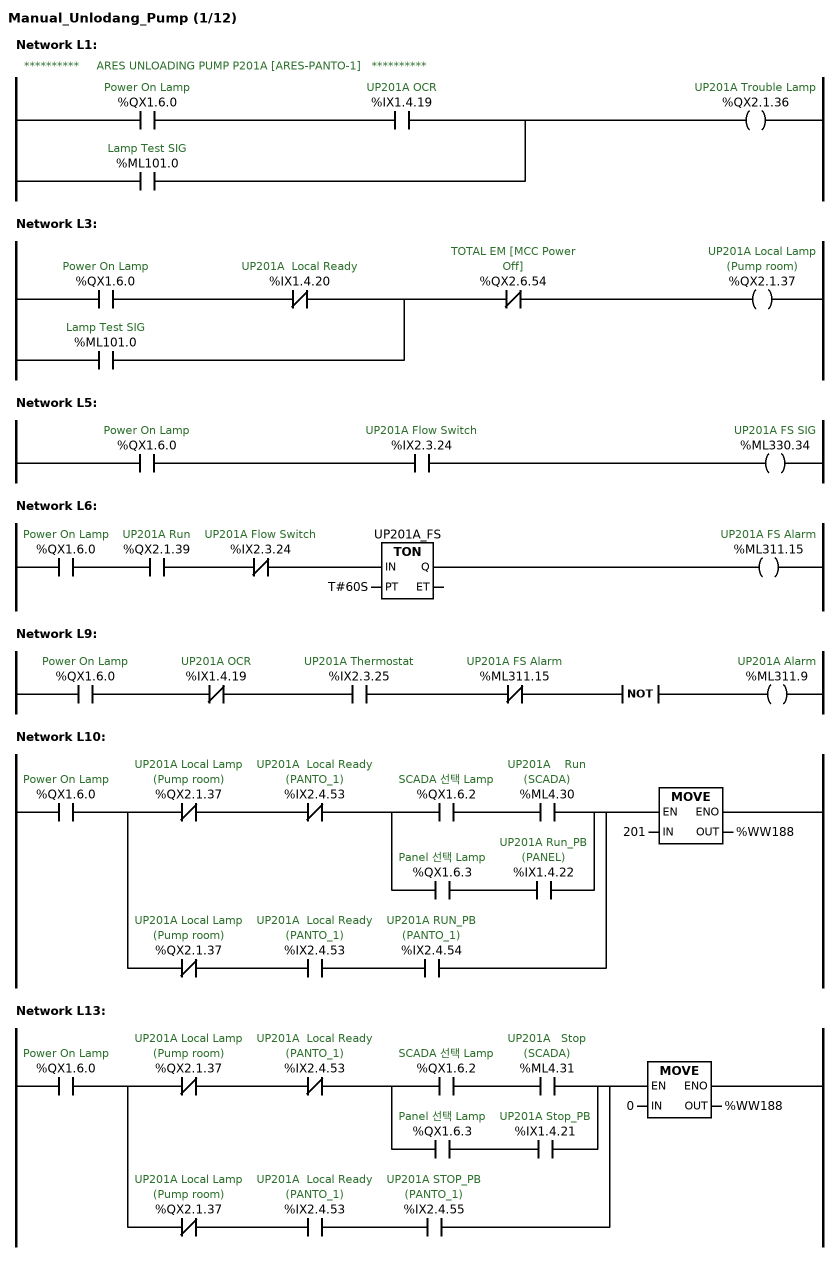
(* **********     ARES UNLOADING PUMP P201A [ARES-PANTO-1]   ********** *)
(* Rung L1 *)
%QX2.1.36 := (%QX1.6.0 AND %IX1.4.19) OR %ML101.0;
(* Rung L3 *)
%QX2.1.37 := ((%QX1.6.0 AND NOT %IX1.4.20) OR %ML101.0) AND NOT %QX2.6.54;
(* Rung L5 *)
%ML330.34 := %QX1.6.0 AND %IX2.3.24;
(* Rung L6 *)
UP201A_FS(IN := %QX1.6.0 AND %QX2.1.39 AND NOT %IX2.3.24, PT := T#60S);
%ML311.15 := UP201A_FS.Q;
(* Rung L9 *)
%ML311.9 := NOT (%QX1.6.0 AND NOT %IX1.4.19 AND %IX2.3.25 AND NOT %ML311.15);
(* Rung L10 *)
IF %QX1.6.0 AND ((NOT %QX2.1.37 AND NOT %IX2.4.53 AND ((%QX1.6.2 AND %ML4.30) OR (%QX1.6.3 AND %IX1.4.22))) OR (NOT %QX2.1.37 AND %IX2.4.53 AND %IX2.4.54)) THEN
    %WW188 := 201;
END_IF;
(* Rung L13 *)
IF %QX1.6.0 AND ((NOT %QX2.1.37 AND NOT %IX2.4.53 AND ((%QX1.6.2 AND %ML4.31) OR (%QX1.6.3 AND %IX1.4.21))) OR (NOT %QX2.1.37 AND %IX2.4.53 AND %IX2.4.55)) THEN
    %WW188 := 0;
END_IF;

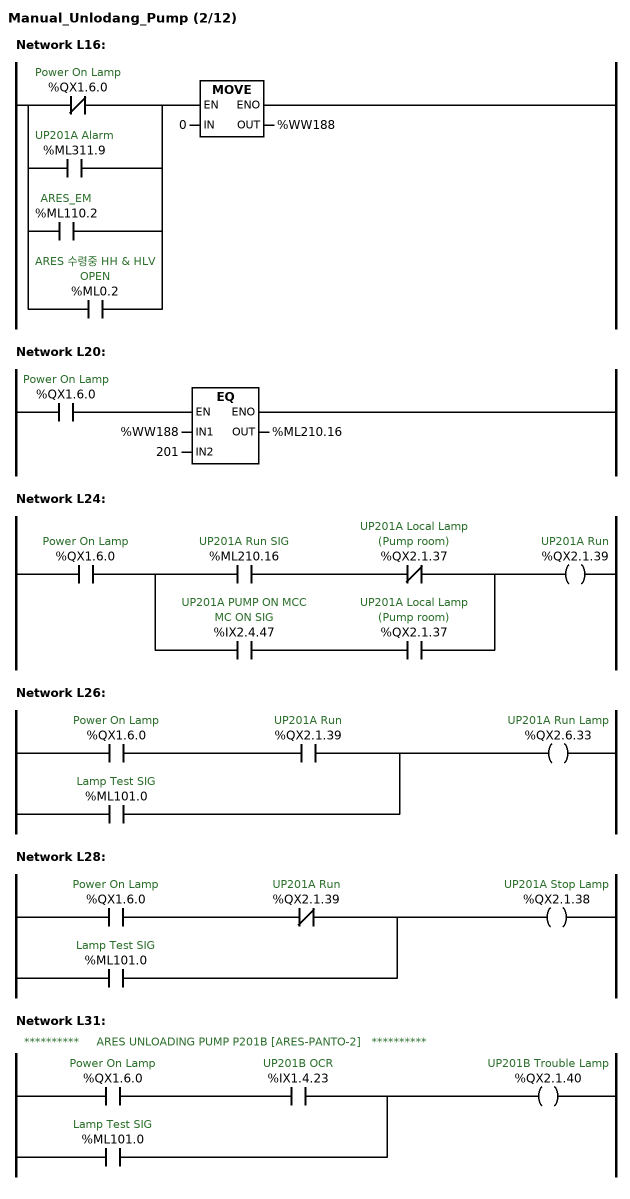
(* Rung L16 *)
IF NOT %QX1.6.0 OR %ML311.9 OR %ML110.2 OR %ML0.2 THEN %WW188 := 0; END_IF;
(* Rung L20 *)
IF %QX1.6.0 THEN %ML210.16 := %WW188 = 201; END_IF;
(* Rung L24 *)
%QX2.1.39 := %QX1.6.0 AND ((%ML210.16 AND NOT %QX2.1.37) OR (%IX2.4.47 AND %QX2.1.37));
(* Rung L26 *)
%QX2.6.33 := (%QX1.6.0 AND %QX2.1.39) OR %ML101.0;
(* Rung L28 *)
%QX2.1.38 := (%QX1.6.0 AND NOT %QX2.1.39) OR %ML101.0;
(* **********     ARES UNLOADING PUMP P201B [ARES-PANTO-2]   ********** *)
(* Rung L31 *)
%QX2.1.40 := (%QX1.6.0 AND %IX1.4.23) OR %ML101.0;

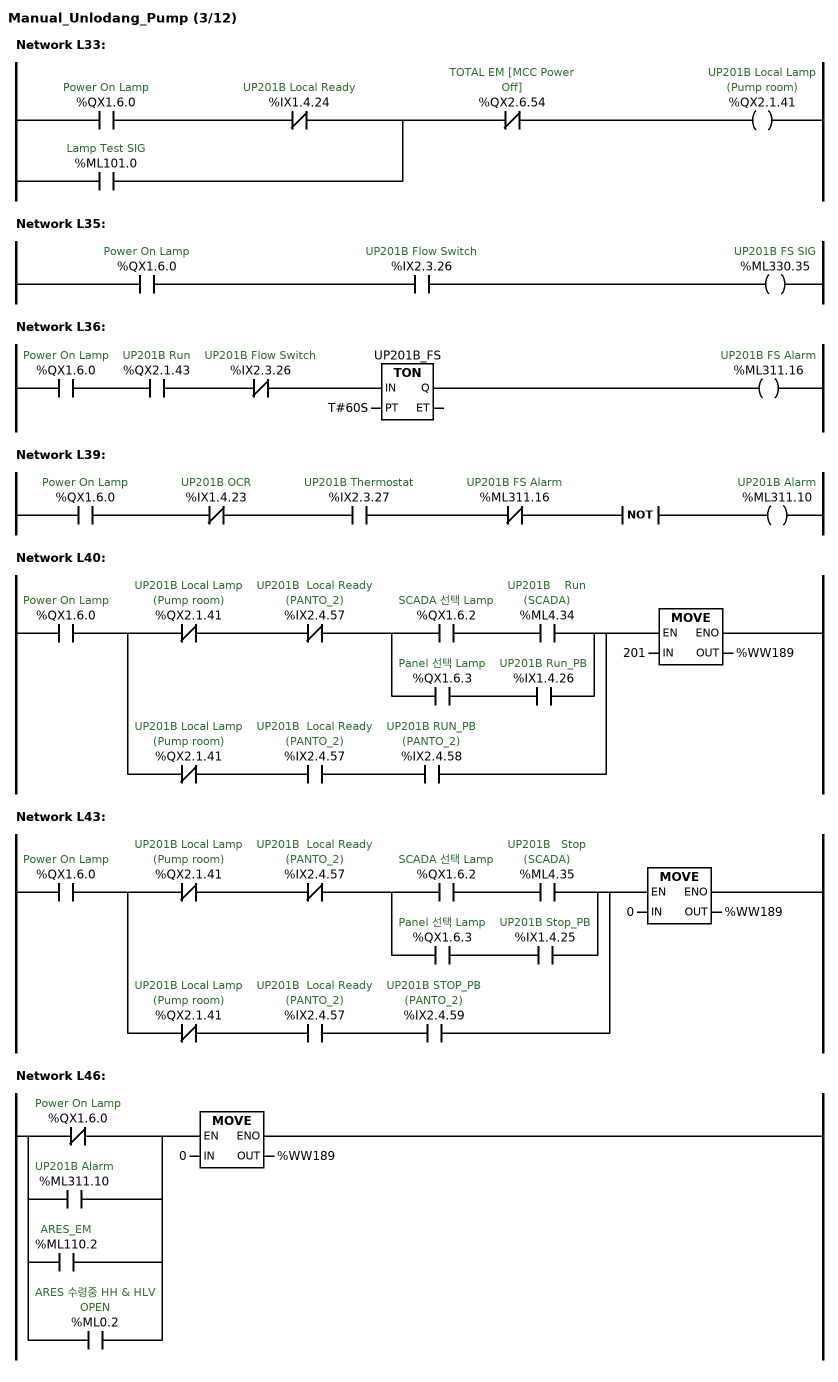
(* Rung L33 *)
%QX2.1.41 := ((%QX1.6.0 AND NOT %IX1.4.24) OR %ML101.0) AND NOT %QX2.6.54;
(* Rung L35 *)
%ML330.35 := %QX1.6.0 AND %IX2.3.26;
(* Rung L36 *)
UP201B_FS(IN := %QX1.6.0 AND %QX2.1.43 AND NOT %IX2.3.26, PT := T#60S);
%ML311.16 := UP201B_FS.Q;
(* Rung L39 *)
%ML311.10 := NOT (%QX1.6.0 AND NOT %IX1.4.23 AND %IX2.3.27 AND NOT %ML311.16);
(* Rung L40 *)
IF %QX1.6.0 AND ((NOT %QX2.1.41 AND NOT %IX2.4.57 AND ((%QX1.6.2 AND %ML4.34) OR (%QX1.6.3 AND %IX1.4.26))) OR (NOT %QX2.1.41 AND %IX2.4.57 AND %IX2.4.58)) THEN
    %WW189 := 201;
END_IF;
(* Rung L43 *)
IF %QX1.6.0 AND ((NOT %QX2.1.41 AND NOT %IX2.4.57 AND ((%QX1.6.2 AND %ML4.35) OR (%QX1.6.3 AND %IX1.4.25))) OR (NOT %QX2.1.41 AND %IX2.4.57 AND %IX2.4.59)) THEN
    %WW189 := 0;
END_IF;
(* Rung L46 *)
IF NOT %QX1.6.0 OR %ML311.10 OR %ML110.2 OR %ML0.2 THEN %WW189 := 0; END_IF;

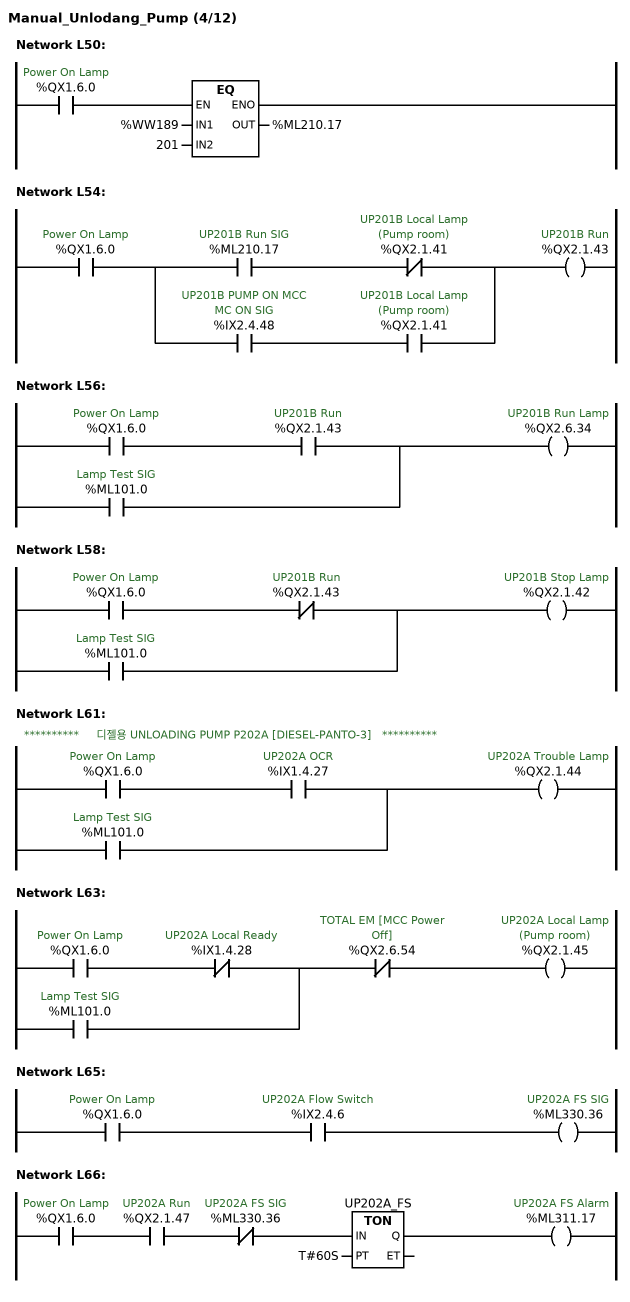
(* Rung L50 *)
IF %QX1.6.0 THEN %ML210.17 := %WW189 = 201; END_IF;
(* Rung L54 *)
%QX2.1.43 := %QX1.6.0 AND ((%ML210.17 AND NOT %QX2.1.41) OR (%IX2.4.48 AND %QX2.1.41));
(* Rung L56 *)
%QX2.6.34 := (%QX1.6.0 AND %QX2.1.43) OR %ML101.0;
(* Rung L58 *)
%QX2.1.42 := (%QX1.6.0 AND NOT %QX2.1.43) OR %ML101.0;
(* **********     디젤용 UNLOADING PUMP P202A [DIESEL-PANTO-3]   ********** *)
(* Rung L61 *)
%QX2.1.44 := (%QX1.6.0 AND %IX1.4.27) OR %ML101.0;
(* Rung L63 *)
%QX2.1.45 := ((%QX1.6.0 AND NOT %IX1.4.28) OR %ML101.0) AND NOT %QX2.6.54;
(* Rung L65 *)
%ML330.36 := %QX1.6.0 AND %IX2.4.6;
(* Rung L66 *)
UP202A_FS(IN := %QX1.6.0 AND %QX2.1.47 AND NOT %ML330.36, PT := T#60S);
%ML311.17 := UP202A_FS.Q;

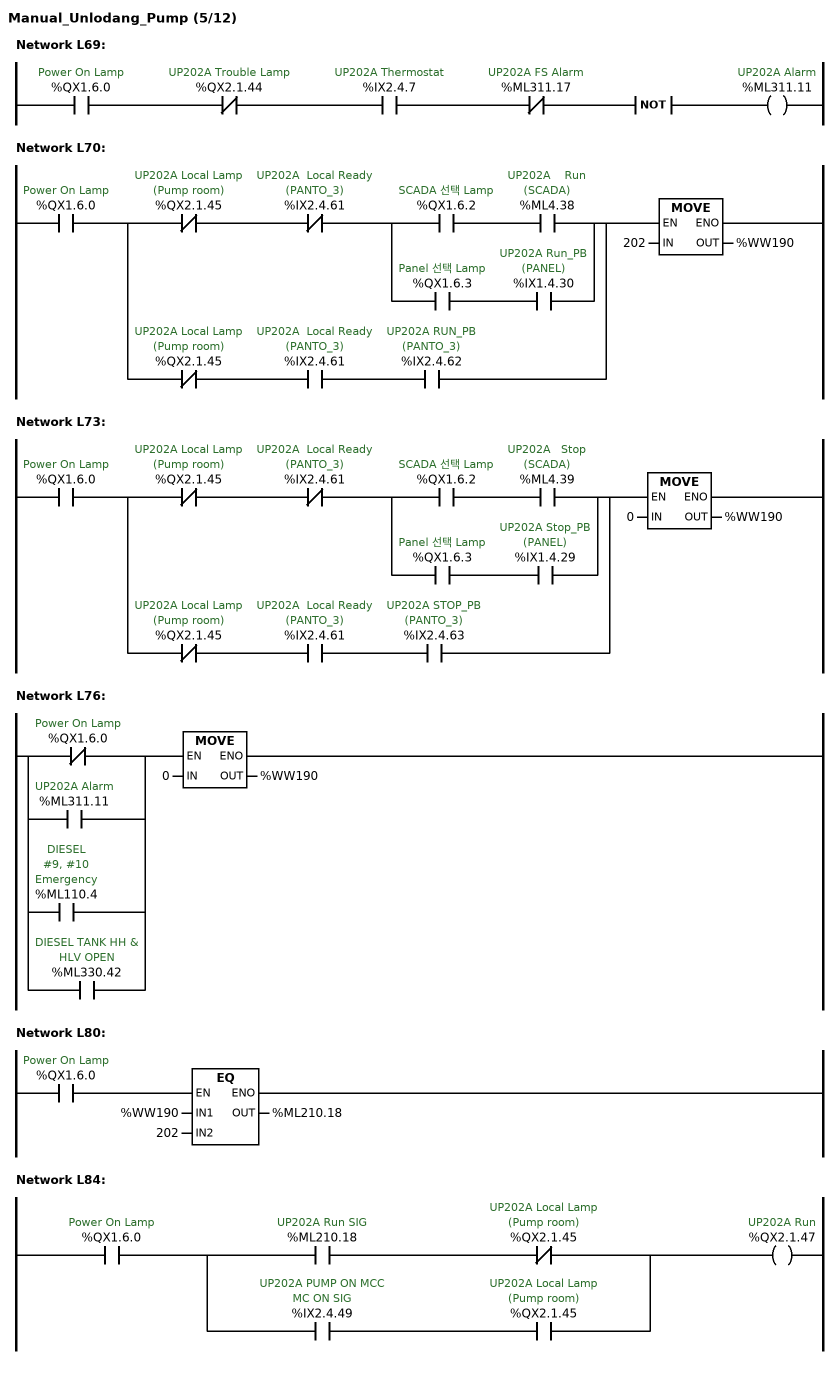
(* Rung L69 *)
%ML311.11 := NOT (%QX1.6.0 AND NOT %QX2.1.44 AND %IX2.4.7 AND NOT %ML311.17);
(* Rung L70 *)
IF %QX1.6.0 AND ((NOT %QX2.1.45 AND NOT %IX2.4.61 AND ((%QX1.6.2 AND %ML4.38) OR (%QX1.6.3 AND %IX1.4.30))) OR (NOT %QX2.1.45 AND %IX2.4.61 AND %IX2.4.62)) THEN
    %WW190 := 202;
END_IF;
(* Rung L73 *)
IF %QX1.6.0 AND ((NOT %QX2.1.45 AND NOT %IX2.4.61 AND ((%QX1.6.2 AND %ML4.39) OR (%QX1.6.3 AND %IX1.4.29))) OR (NOT %QX2.1.45 AND %IX2.4.61 AND %IX2.4.63)) THEN
    %WW190 := 0;
END_IF;
(* Rung L76 *)
IF NOT %QX1.6.0 OR %ML311.11 OR %ML110.4 OR %ML330.42 THEN %WW190 := 0; END_IF;
(* Rung L80 *)
IF %QX1.6.0 THEN %ML210.18 := %WW190 = 202; END_IF;
(* Rung L84 *)
%QX2.1.47 := %QX1.6.0 AND ((%ML210.18 AND NOT %QX2.1.45) OR (%IX2.4.49 AND %QX2.1.45));

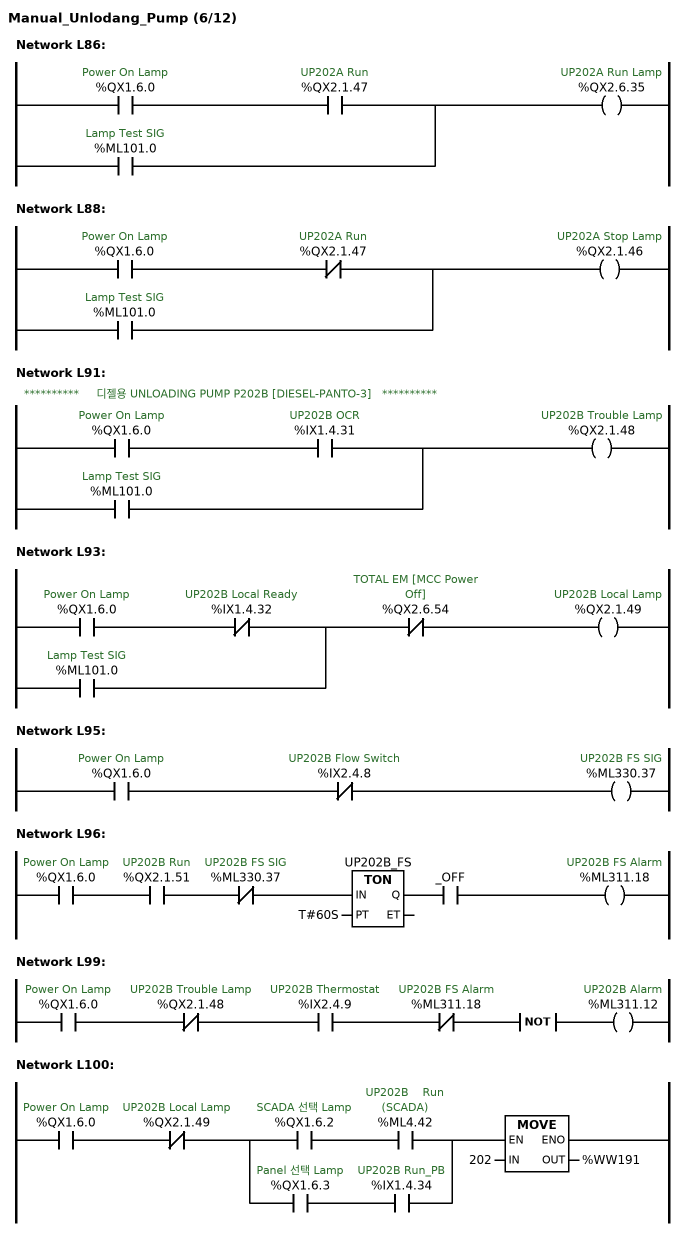
(* Rung L86 *)
%QX2.6.35 := (%QX1.6.0 AND %QX2.1.47) OR %ML101.0;
(* Rung L88 *)
%QX2.1.46 := (%QX1.6.0 AND NOT %QX2.1.47) OR %ML101.0;
(* **********     디젤용 UNLOADING PUMP P202B [DIESEL-PANTO-3]   ********** *)
(* Rung L91 *)
%QX2.1.48 := (%QX1.6.0 AND %IX1.4.31) OR %ML101.0;
(* Rung L93 *)
%QX2.1.49 := ((%QX1.6.0 AND NOT %IX1.4.32) OR %ML101.0) AND NOT %QX2.6.54;
(* Rung L95 *)
%ML330.37 := %QX1.6.0 AND NOT %IX2.4.8;
(* Rung L96 *)
UP202B_FS(IN := %QX1.6.0 AND %QX2.1.51 AND NOT %ML330.37, PT := T#60S);
%ML311.18 := UP202B_FS.Q AND _OFF;
(* Rung L99 *)
%ML311.12 := NOT (%QX1.6.0 AND NOT %QX2.1.48 AND %IX2.4.9 AND NOT %ML311.18);
(* Rung L100 *)
IF %QX1.6.0 AND NOT %QX2.1.49 AND ((%QX1.6.2 AND %ML4.42) OR (%QX1.6.3 AND %IX1.4.34)) THEN
    %WW191 := 202;
END_IF;

